(* PLC project Unnamed, Unknown Unnamed 1 *)
(* stored: creationDateTime 2026-09-05T12:24:49, modificationDateTime 2026-09-05T12:24:49 *)

FUNCTION_BLOCK CTU
  VAR_OUTPUT
    Q : BOOL;
    CV : INT;
  END_VAR
  VAR_INPUT
    CU : BOOL;
    R : BOOL;
    PV : INT;
  END_VAR

END_FUNCTION_BLOCK

FUNCTION GE : BOOL
  VAR_INPUT
    IN1 : ANY_ELEMENTARY;
    IN2 : ANY_ELEMENTARY;
  END_VAR

END_FUNCTION

FUNCTION LE : BOOL
  VAR_INPUT
    IN1 : ANY_ELEMENTARY;
    IN2 : ANY_ELEMENTARY;
  END_VAR

END_FUNCTION

FUNCTION MOVE : ANY
  VAR_INPUT
    IN : ANY;
  END_VAR

END_FUNCTION

FUNCTION_BLOCK R_TRIG
  VAR_OUTPUT
    Q : BOOL;
  END_VAR
  VAR_INPUT
    CLK : BOOL;
  END_VAR

END_FUNCTION_BLOCK

FUNCTION_BLOCK SR
  VAR_OUTPUT
    Q1 : BOOL;
  END_VAR
  VAR_INPUT
    S1 : BOOL;
    R : BOOL;
  END_VAR

END_FUNCTION_BLOCK

FUNCTION_BLOCK TON
  VAR_OUTPUT
    Q : BOOL;
    ET : TIME;
  END_VAR
  VAR_INPUT
    IN : BOOL;
    PT : TIME;
  END_VAR

END_FUNCTION_BLOCK

(* VARIABLES TABLE *)
PROGRAM automated_conveyor_sorting_and_batching_system
  VAR
    START_PB AT %IX0.0 : BOOL := FALSE;  (* START BUTTON *)
    STOP_PB AT %IX0.1 : BOOL := FALSE;  (* STOP BUTTON *)
    ESTOP_OK AT %IX0.2 : BOOL := FALSE;  (* E-STOP HEALTHY *)
    OVRLOAD_OK AT %IX0.3 : BOOL := FALSE;  (* OVERLOAD HEALTHY *)
    MOTOR_RUN AT %QX0.0 : BOOL;  (* MOTOR OUTPUT *)
    LAMP_RUN AT %QX0.1 : BOOL;  (* RUNNING INDICATOR *)
    PRODUCT_SENSOR AT %IX0.4 : BOOL := FALSE;  (* DETECTING PRODUCTS *)
    REJECT_SELENOID AT %QX0.2 : BOOL := FALSE;  (* Actuator to reject non-standard products *)
    QUALITY_SENSOR AT %IX0.5 : BOOL;  (* Sensor ascertaining Quality other than weight *)
    BATCH_RESET_PB AT %MX0.2 : BOOL;  (* Counter reset button *)
    BATCH_COMPLETE_LAMP AT %QX0.3 : BOOL;  (* Process completion indicator *)
    RAW_WEIGHT AT %IW0 : INT := 0;  (* Raw integer reading from the scale's analog channel(0 - 32767) *)
    ACTUAL_WEIGHT AT %MD0 : REAL := 0.0;  (* Calculated real weight of the product in kgs *)
    MIN_WEIGHT AT %MD2 : REAL := 49.95;  (* Lower allowed limit *)
    MAX_WEIGHT AT %MD4 : REAL := 50.10;  (* Upper allowed limit *)
    WEIGHT_OK AT %QX0.4 : BOOL := FALSE;  (* Internal flag: TRUE when weight is valid *)
    HMI_MOTOR_CMD AT %MX0.0 : BOOL;  (* Start command triggered from HMI *)
    HMI_STOP_CMD AT %MX0.1 : BOOL;  (* Stop command triggered from HMI *)
    BATCH_COUNT_VALUE AT %MW0 : INT := 0;  (* Displays incrementaly the Batch count *)
  END_VAR
  VAR
    SR0 : SR;  (* Memory block *)
    TON1 : TON;  (* Product Travel time Timer *)
    R_TRIG0 : R_TRIG;  (* Rising Edge Trigger *)
    TON2 : TON;  (* Actuator reset Timer *)
    R_TRIG1 : R_TRIG;  (* Rising Edge Trigger *)
    CTU1 : CTU;  (* UP Counter for incrementing detected allowed products *)
    TON3 : TON;  (* UP Counter reset Timer *)
    RAW_REAL : REAL := 0.0;  (* Temporary Floating_point values for maths *)
    SCALE_FACTOR : REAL := 0.00152588;  (* Coversion multiplier max kg/max raw = 50.0/32767.0 *)
    ABOVE_MIN : BOOL;  (* GE Block Boolean output *)
    BELOW_MAX : BOOL;  (* LE Boolean output *)
    INIT_BIT : BOOL := FALSE;
  END_VAR
  VAR  (* added by the conversion: wires and edge detectors of the diagram *)
    _MOVE8751718_ENO : BOOL;
    _MOVE8751718_OUT : ANY;
    _MOVE3884773_ENO : BOOL;
    _MOVE3884773_OUT : ANY;
    _GE10858314_ENO : BOOL;
    _GE10858314_OUT : BOOL;
    _LE5869513_ENO : BOOL;
    _LE5869513_OUT : BOOL;
  END_VAR

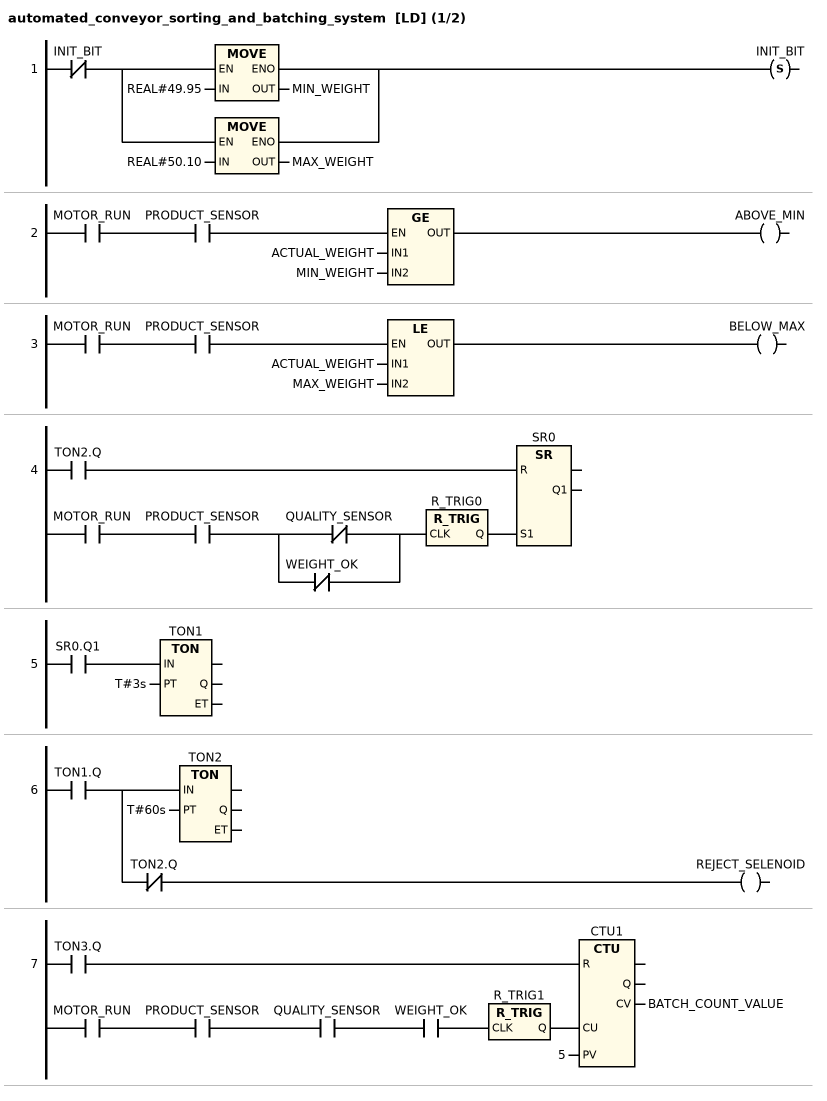
(* LD diagram, written out as Structured Text *)
IF HMI_STOP_CMD THEN HMI_MOTOR_CMD := FALSE; END_IF;
IF HMI_STOP_CMD THEN MOTOR_RUN := FALSE; END_IF;
MOTOR_RUN := NOT STOP_PB AND NOT HMI_STOP_CMD AND NOT ESTOP_OK AND NOT OVRLOAD_OK AND (START_PB OR HMI_MOTOR_CMD OR MOTOR_RUN);
MOTOR_RUN := NOT STOP_PB AND NOT ESTOP_OK AND NOT OVRLOAD_OK AND HMI_MOTOR_CMD;
LAMP_RUN := MOTOR_RUN;
_MOVE8751718_OUT := MOVE(EN := NOT INIT_BIT, IN := REAL#49.95, ENO => _MOVE8751718_ENO);
_MOVE3884773_OUT := MOVE(EN := NOT INIT_BIT, IN := REAL#50.10, ENO => _MOVE3884773_ENO);
IF _MOVE8751718_ENO OR _MOVE3884773_ENO THEN INIT_BIT := TRUE; END_IF;
_GE10858314_OUT := GE(EN := MOTOR_RUN AND PRODUCT_SENSOR, IN1 := ACTUAL_WEIGHT, IN2 := MIN_WEIGHT, ENO => _GE10858314_ENO);
ABOVE_MIN := _GE10858314_OUT;
_LE5869513_OUT := LE(EN := MOTOR_RUN AND PRODUCT_SENSOR, IN1 := ACTUAL_WEIGHT, IN2 := MAX_WEIGHT, ENO => _LE5869513_ENO);
BELOW_MAX := _LE5869513_OUT;
WEIGHT_OK := MOTOR_RUN AND PRODUCT_SENSOR AND ABOVE_MIN AND BELOW_MAX;
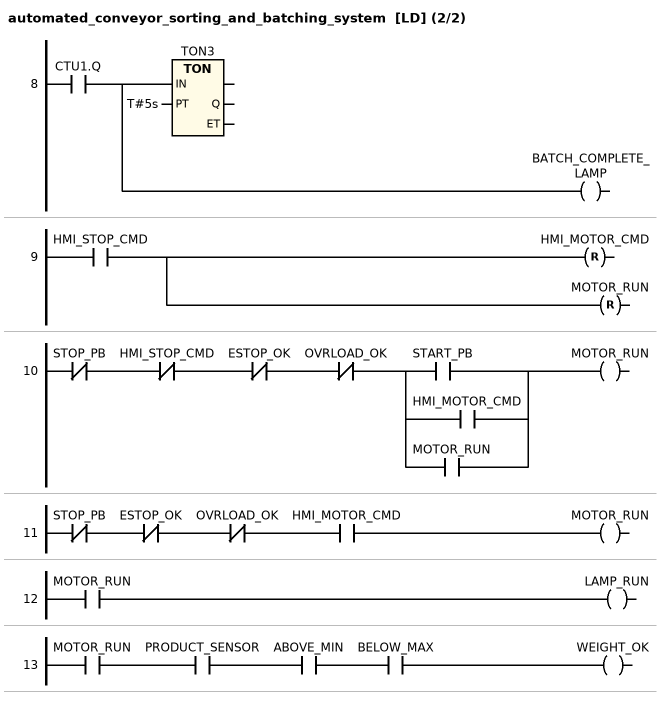
REJECT_SELENOID := TON1.Q AND NOT TON2.Q;
BATCH_COMPLETE_LAMP := CTU1.Q;
IF _MOVE8751718_ENO THEN MIN_WEIGHT := _MOVE8751718_OUT; END_IF;
IF _MOVE3884773_ENO THEN MAX_WEIGHT := _MOVE3884773_OUT; END_IF;
TON1(IN := SR0.Q1, PT := T#3s);
 := TON1.ET;
TON2(IN := TON1.Q, PT := T#60s);
 := TON2.ET;
R_TRIG1(CLK := MOTOR_RUN AND PRODUCT_SENSOR AND QUALITY_SENSOR AND WEIGHT_OK);
CTU1(CU := R_TRIG1.Q, R := TON3.Q, PV := 5);
BATCH_COUNT_VALUE := CTU1.CV;
TON3(IN := CTU1.Q, PT := T#5s);
 := TON3.ET;
R_TRIG0(CLK := MOTOR_RUN AND PRODUCT_SENSOR AND (NOT QUALITY_SENSOR OR NOT WEIGHT_OK));
SR0(S1 := R_TRIG0.Q, R := TON2.Q);
END_PROGRAM

CONFIGURATION Config0
  RESOURCE Res0 ON PLC
    TASK task1(INTERVAL := T#20ms, PRIORITY := 1);
    PROGRAM instance1 WITH task1 : automated_conveyor_sorting_and_batching_system;
  END_RESOURCE
END_CONFIGURATION
